{attribute 'qualified_only'}
VAR_GLOBAL
END_VAR

(* stored: Version 1.1.0.1, ProductVersion 3.1.4024.13
   GVL Outputs: Id {55043a6e-9b53-461d-9f9c-c0a1d203dd65} *)
